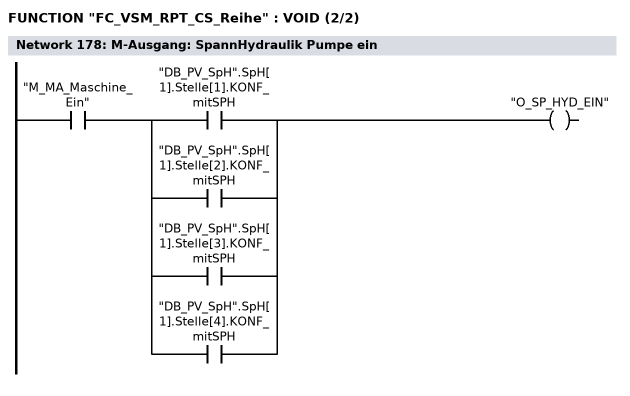

      U     "M_MA_Maschine_Ein";
      U(    ;
      O     "DB_PV_SpH".SpH[1].Stelle[1].KONF_mitSPH;
      O     "DB_PV_SpH".SpH[1].Stelle[2].KONF_mitSPH;
      O     "DB_PV_SpH".SpH[1].Stelle[3].KONF_mitSPH;
      O     "DB_PV_SpH".SpH[1].Stelle[4].KONF_mitSPH;
      )     ;
      =     "O_SP_HYD_EIN";
NETWORK
TITLE =Aufruf: Rüstplatztüre entriegeln

RPT:  CALL "FC_RPT_ENTRIEGELN" ;
      NOP   0;
END_FUNCTION

